PROGRAM Communications
VAR
END_VAR

END_PROGRAM

(* stored: Version 1.1.0.1, ProductVersion 3.1.4024.12
   POU Communications: Id {7df06c8f-9929-4624-86ed-db6de593a22b}, SpecialFunc None *)
